TYPE ST_SCANNER_ImageData :
STRUCT
	nCodesRead		: INT;
	tScanTime		: TIME;		(* image cycle time (including image acquisition time and decode time) *)
	sStatus			: T_MaxString;
	stTriggerID		: ST_SCANNER_TriggerID;
	aCodeData		: ARRAY[1..cMAX_CAMERA_PROG_NUMBER] OF ST_SCANNER_CodeData;
END_STRUCT
END_TYPE

(* stored: Version 1.1.0.1, ProductVersion 3.1.4024.15
   DUT ST_SCANNER_ImageData: Id {4856edd7-2e4c-4fa8-ab37-5891843cd423} *)
